PROGRAM FC2
VAR
END_VAR

END_PROGRAM

(* stored: Version 1.1.0.1, ProductVersion 3.1.4022.12
   POU FC2: Id {6d3fc48b-8611-4990-8b52-215656a9b975}, SpecialFunc None *)
